# EPICS substitutions: devel/epics/drivers/jlabVMEBoardApp/Db/user.substitutions
# Example substitutions file

file "db/dbExample1.db" {
    { user = "hovanes" }
}

file db/dbExample2.db {
    pattern { user, no, scan }
        { "hovanes", 1, "1 second" }
        { "hovanes", 2, "2 second" }
        { "hovanes", 3, "5 second" }
}
